PROGRAM MAIN
VAR
END_VAR

END_PROGRAM

(* stored: Version 1.1.0.1
   POU MAIN: Id {71f160f7-3e2f-447b-b103-83a6cae327b2} *)
